/// Use of this pattern is *NOT* recommended 
FUNCTION_BLOCK FbFlasher
VAR
	/// pattern original 
	Timer1: Ton;
	tET1: TIME;
	Timer2: Ton;
	tET2: TIME;
	/// IEC standard alternative 
	BLINK: util.BLINK;
	xBlink: BOOL;
END_VAR
VAR_OUTPUT
	xFlashingLight: BOOL;
END_VAR

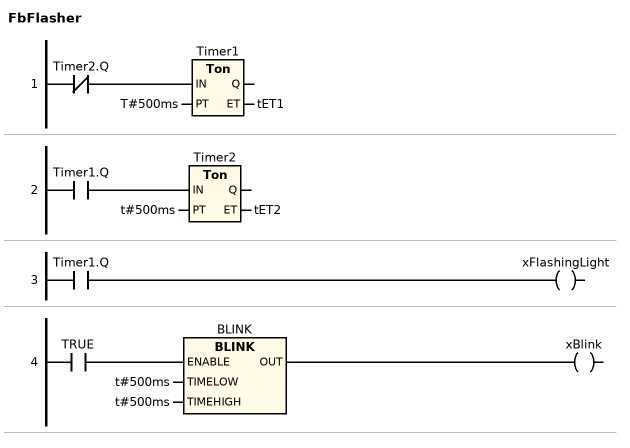
// NETWORK 1
Timer1(IN := NOT Timer2.Q, PT := T#500ms, ET => tET1); // Ton

// NETWORK 2
Timer2(IN := Timer1.Q, PT := t#500ms, ET => tET2); // Ton

// NETWORK 3
xFlashingLight := Timer1.Q;

// NETWORK 4
BLINK(ENABLE := TRUE, TIMELOW := t#500ms, TIMEHIGH := t#500ms);
xBlink := BLINK.OUT;

END_FUNCTION_BLOCK

(* stored: Version 1.1.0.1, ProductVersion 3.1.4024.12
   POU FbFlasher: Id {e2a492c3-4bb0-4b19-a886-54fe8ab99b32}, SpecialFunc None *)
